Fanuc TP program (LS listing): PTPROBE.LS

/PROG  PTPROBE
/ATTR
OWNER		= MNEDITOR;
COMMENT		= "point probe";
PROG_SIZE	= 0;
CREATE		= DATE 26-01-01  TIME 00:00:00;
MODIFIED	= DATE 26-01-01  TIME 00:00:00;
FILE_NAME	= ;
VERSION		= 0;
LINE_COUNT	= 18;
MEMORY_SIZE	= 0;
PROTECT		= READ_WRITE;
TCD:  STACK_SIZE	= 0,
      TASK_PRIORITY	= 50,
      TIME_SLICE	= 0,
      BUSY_LAMP_OFF	= 0,
      ABORT_REQUEST	= 0,
      PAUSE_REQUEST	= 0;
DEFAULT_GROUP	= 1,*,*,*,*;
CONTROL_CODE	= 00000000 00000000;
/MN
   1:  !CrossArm point probe ;
   2:  PR[100]=P[1]    ;
   3:  UTOOL[1]=PR[100] ;
   4:  PR[100]=P[2]    ;
   5:  UFRAME[1]=PR[100] ;
   6:  PR[90]=P[3]    ;
   7:  PR[91]=P[4]    ;
   8:  PR[92]=P[5]    ;
   9:  PR[93]=P[6]    ;
  10:  PR[49]=P[7]    ;
  11:  UTOOL[9]=PR[49] ;
  12:  UFRAME_NUM=0 ;
  13:  UTOOL_NUM=9 ;
  14:J P[8] 10% FINE    ;
  15:  R[90]=1    ;
  16:  CALL POINTPROBE    ;
  17:  R[90]=46    ;
  18:  CALL POINTDIRECT    ;
/POS
P[1]{
   GP1:
	UF : 0, UT : 1,		CONFIG : 'N U T, 0, 0, 0',
	X =    10.000  mm,	Y =    -5.000  mm,	Z =   120.000  mm,
	W =     0.000 deg,	P =     0.000 deg,	R =     0.000 deg
};
P[2]{
   GP1:
	UF : 0, UT : 1,		CONFIG : 'N U T, 0, 0, 0',
	X =  1100.000  mm,	Y =  -150.000  mm,	Z =   650.000  mm,
	W =     0.000 deg,	P =     0.000 deg,	R =    10.000 deg
};
P[3]{
   GP1:
	UF : 0, UT : 1,		CONFIG : 'N U T, 0, 0, 0',
	X =    40.000  mm,	Y =   -40.000  mm,	Z =   230.000  mm,
	W =   180.000 deg,	P =     0.000 deg,	R =     0.000 deg
};
P[4]{
   GP1:
	UF : 0, UT : 1,		CONFIG : 'N U T, 0, 0, 0',
	X =   100.000  mm,	Y =   -40.000  mm,	Z =   230.000  mm,
	W =   180.000 deg,	P =     0.000 deg,	R =     0.000 deg
};
P[5]{
   GP1:
	UF : 0, UT : 1,		CONFIG : 'N U T, 0, 0, 0',
	X =    40.000  mm,	Y =    60.000  mm,	Z =   230.000  mm,
	W =   180.000 deg,	P =     0.000 deg,	R =     0.000 deg
};
P[6]{
   GP1:
	UF : 0, UT : 1,		CONFIG : 'N U T, 0, 0, 0',
	X =   100.000  mm,	Y =    60.000  mm,	Z =   230.000  mm,
	W =   180.000 deg,	P =     0.000 deg,	R =     0.000 deg
};
P[7]{
   GP1:
	UF : 0, UT : 1,		CONFIG : 'N U T, 0, 0, 0',
	X =     0.000  mm,	Y =     0.000  mm,	Z =     0.000  mm,
	W =     0.000 deg,	P =     0.000 deg,	R =     0.000 deg
};
P[8]{
   GP1:
	UF : 0, UT : 9,
	J1=     0.000 deg,	J2=     0.000 deg,	J3=     0.000 deg,
	J4=     0.000 deg,	J5=   -90.000 deg,	J6=     0.000 deg
};
/END
